// Mitsubishi GX Works2 project: plc+hmi2+   PLC: Q03UDV

PROGRAM MAIN
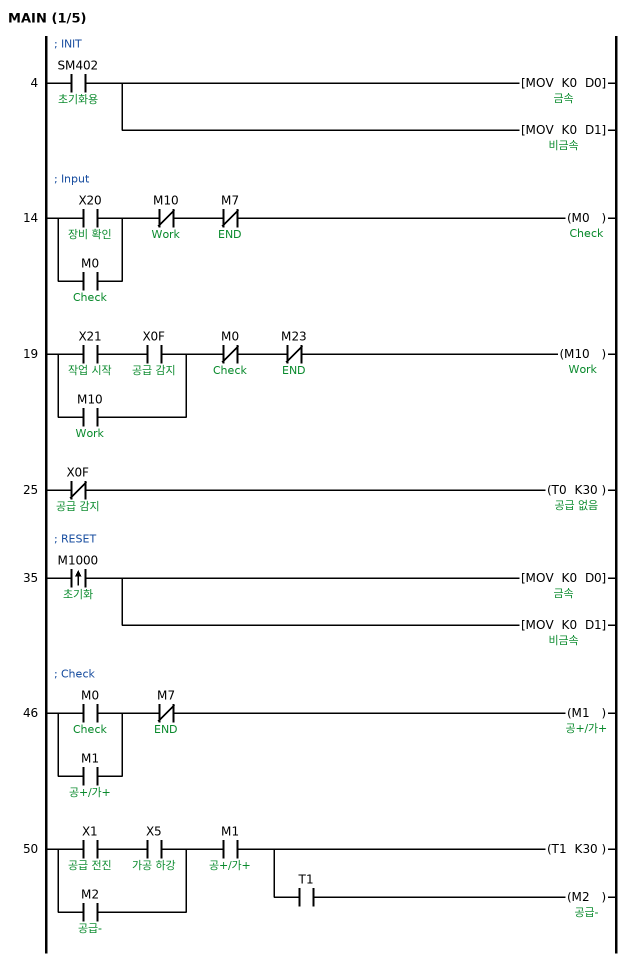
; INIT
4     LD      SM402  ; 초기화용
      MOV     K0 D0  ; 금속
      MOV     K0 D1  ; 비금속
; Input
14    LD      X20  ; 장비 확인
      OR      M0  ; Check
      ANI     M10  ; Work
      ANI     M7  ; END
      OUT     M0  ; Check
19    LD      X21  ; 작업 시작
      AND     X0F  ; 공급 감지
      OR      M10  ; Work
      ANI     M0  ; Check
      ANI     M23  ; END
      OUT     M10  ; Work
25    LDI     X0F  ; 공급 감지
      OUT     T0 K30  ; 공급 없음
; RESET
35    LDP     M1000  ; 초기화
      MOV     K0 D0
      MOV     K0 D1
; Check
46    LD      M0  ; Check
      OR      M1  ; 공+/가+
      ANI     M7  ; END
      OUT     M1  ; 공+/가+
50    LD      X1  ; 공급 전진
      AND     X5  ; 가공 하강
      OR      M2  ; 공급-
      AND     M1  ; 공+/가+
      OUT     T1 K30
      AND     T1
      OUT     M2  ; 공급-
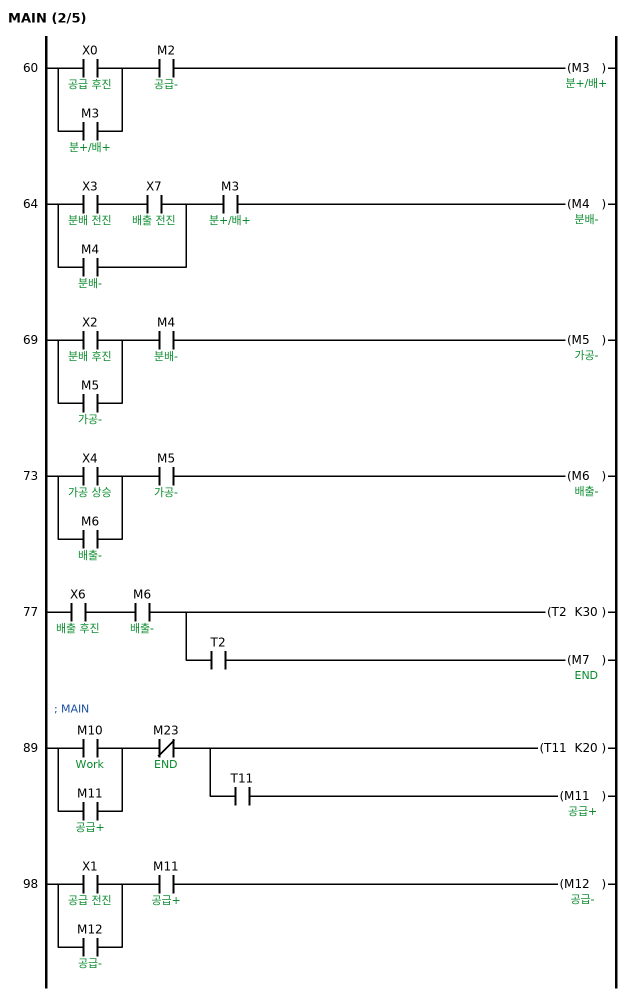
60    LD      X0  ; 공급 후진
      OR      M3  ; 분+/배+
      AND     M2  ; 공급-
      OUT     M3  ; 분+/배+
64    LD      X3  ; 분배 전진
      AND     X7  ; 배출 전진
      OR      M4  ; 분배-
      AND     M3  ; 분+/배+
      OUT     M4  ; 분배-
69    LD      X2  ; 분배 후진
      OR      M5  ; 가공-
      AND     M4  ; 분배-
      OUT     M5  ; 가공-
73    LD      X4  ; 가공 상승
      OR      M6  ; 배출-
      AND     M5  ; 가공-
      OUT     M6  ; 배출-
77    LD      X6  ; 배출 후진
      AND     M6  ; 배출-
      OUT     T2 K30
      AND     T2
      OUT     M7  ; END
; MAIN
89    LD      M10  ; Work
      OR      M11  ; 공급+
      ANI     M23  ; END
      OUT     T11 K20
      AND     T11
      OUT     M11  ; 공급+
98    LD      X1  ; 공급 전진
      OR      M12  ; 공급-
      AND     M11  ; 공급+
      OUT     M12  ; 공급-
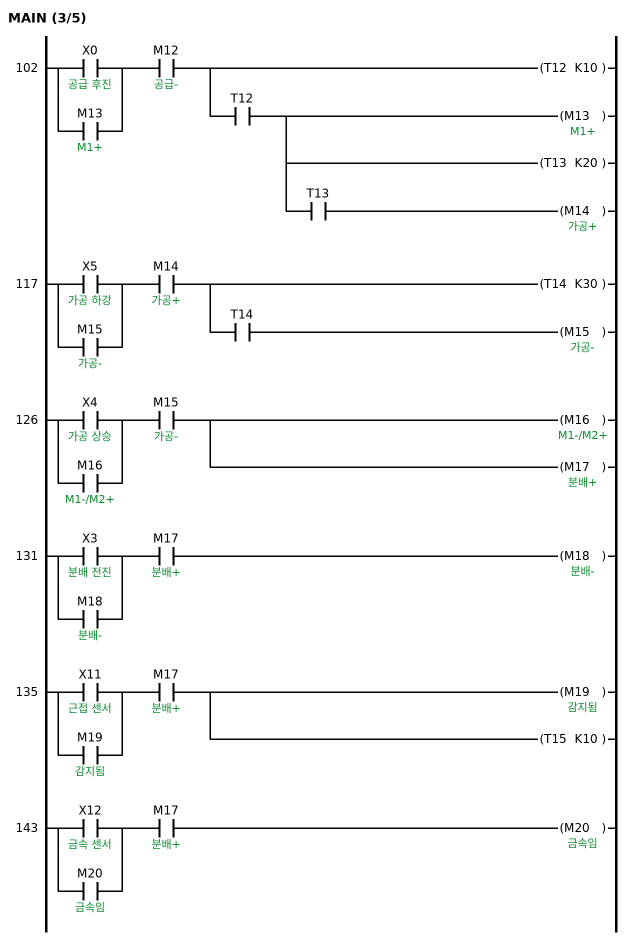
102   LD      X0  ; 공급 후진
      OR      M13  ; M1+
      AND     M12  ; 공급-
      OUT     T12 K10
      AND     T12
      OUT     M13  ; M1+
      OUT     T13 K20
      AND     T13
      OUT     M14  ; 가공+
117   LD      X5  ; 가공 하강
      OR      M15  ; 가공-
      AND     M14  ; 가공+
      OUT     T14 K30
      AND     T14
      OUT     M15  ; 가공-
126   LD      X4  ; 가공 상승
      OR      M16  ; M1-/M2+
      AND     M15  ; 가공-
      OUT     M16  ; M1-/M2+
      OUT     M17  ; 분배+
131   LD      X3  ; 분배 전진
      OR      M18  ; 분배-
      AND     M17  ; 분배+
      OUT     M18  ; 분배-
135   LD      X11  ; 근접 센서
      OR      M19  ; 감지됨
      AND     M17  ; 분배+
      OUT     M19  ; 감지됨
      OUT     T15 K10
143   LD      X12  ; 금속 센서
      OR      M20  ; 금속임
      AND     M17  ; 분배+
      OUT     M20  ; 금속임
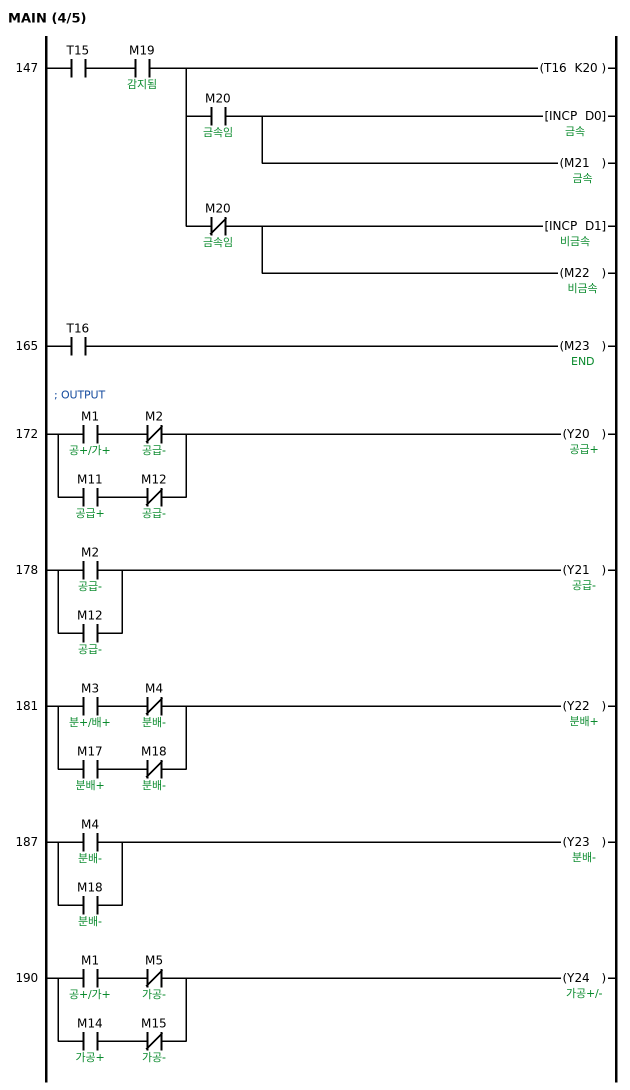
147   LD      T15
      AND     M19  ; 감지됨
      OUT     T16 K20
      MPS
      AND     M20  ; 금속임
      INCP    D0
      OUT     M21  ; 금속
      MPP
      ANI     M20  ; 금속임
      INCP    D1
      OUT     M22  ; 비금속
165   LD      T16
      OUT     M23  ; END
; OUTPUT
172   LD      M1  ; 공+/가+
      ANI     M2  ; 공급-
      LD      M11  ; 공급+
      ANI     M12  ; 공급-
      ORB
      OUT     Y20  ; 공급+
178   LD      M2  ; 공급-
      OR      M12  ; 공급-
      OUT     Y21  ; 공급-
181   LD      M3  ; 분+/배+
      ANI     M4  ; 분배-
      LD      M17  ; 분배+
      ANI     M18  ; 분배-
      ORB
      OUT     Y22  ; 분배+
187   LD      M4  ; 분배-
      OR      M18  ; 분배-
      OUT     Y23  ; 분배-
190   LD      M1  ; 공+/가+
      ANI     M5  ; 가공-
      LD      M14  ; 가공+
      ANI     M15  ; 가공-
      ORB
      OUT     Y24  ; 가공+/-
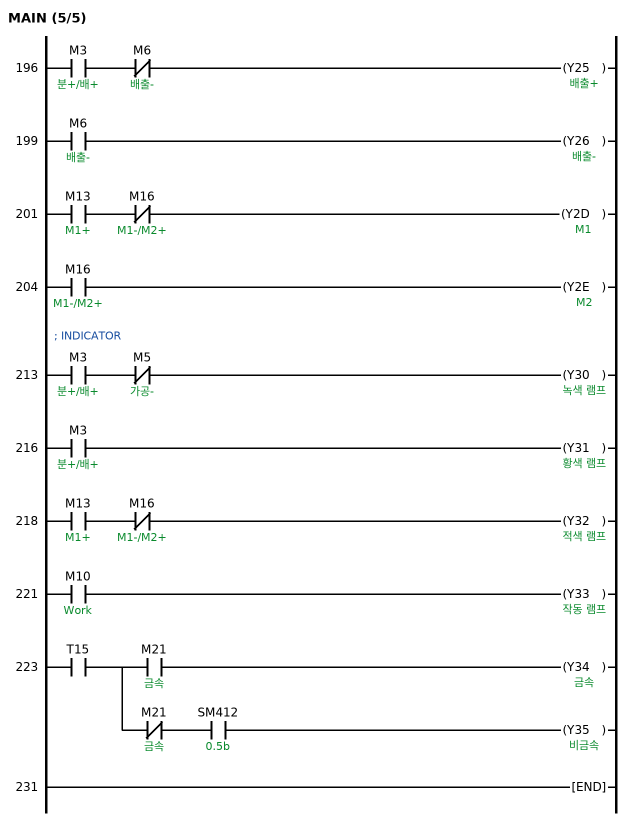
196   LD      M3  ; 분+/배+
      ANI     M6  ; 배출-
      OUT     Y25  ; 배출+
199   LD      M6  ; 배출-
      OUT     Y26  ; 배출-
201   LD      M13  ; M1+
      ANI     M16  ; M1-/M2+
      OUT     Y2D  ; M1
204   LD      M16  ; M1-/M2+
      OUT     Y2E  ; M2
; INDICATOR
213   LD      M3  ; 분+/배+
      ANI     M5  ; 가공-
      OUT     Y30  ; 녹색 램프
216   LD      M3  ; 분+/배+
      OUT     Y31  ; 황색 램프
218   LD      M13  ; M1+
      ANI     M16  ; M1-/M2+
      OUT     Y32  ; 적색 램프
221   LD      M10  ; Work
      OUT     Y33  ; 작동 램프
223   LD      T15
      MPS
      AND     M21  ; 금속
      OUT     Y34  ; 금속
      MPP
      ANI     M21  ; 금속
      AND     SM412  ; 0.5b
      OUT     Y35  ; 비금속
231   END
END_PROGRAM

// device comments not shown above
Y36  ; 금속
M201  ; 가공+
M202  ; 가공-
M301  ; 분배+
M302  ; 분배-
D2  ; 총량
T100  ; 소재없음
T107  ; 배출
T108  ; 적재
